(*
Nazwa:			FB_MoveRegister
Opis:			Blok przesuniecia rejestru formatek
Wersja:			v0.3 		
Data:			2018-11-16
Autor:			DP
Urzadzenia:		 
Konfiguracja:	
Info:
- Są dwa rejestry, wejściowy i wyjsciowy (struktury)
- Jezeli rejestr ma np. 6 elementów to za kazdym razem po wykryciu trigera program będzie
	1 wejściowy przesuwał na 1 wolny (nie ma formatki) wyjściowy
	kasował 1 rejestr wejściowy
	przesuwal rejetr wejsciowy 2 na 1(przeniesiony i skasowany), 3 na 2, 4 na 3, 5 na 4, 6 na 5 i kasowal 6wejsciowy
	tym sposobem po 6 trigerach caly rejestr wejsciowy powinien być na wyjsciowym
	np po 3 trigerach na wyjsciowym powinny byc zajete 1 do 3 i na wejsciowym 1 do 3
Błędy:
1 - nie wyszło z pętli for
2 - formatka już jest w rejestrze
Uwagi:
- 
Zmiany:
2018-09-18 Dodano sprawdzanie nasadek
2018-06-14 DP Pierwsza wersja
*)

FUNCTION_BLOCK FB_MoveRegisterCapControl
VAR_INPUT
	bFirstCycle:BOOL;					//Pierwszy cykl, zeby na początku nie wykrywało zbocza opadającego
	bTrigger :BOOL;						// Przesuniecie tablicy o jeden
	tTriggerFilterTimeOn:TIME:=T#0MS;	// Czas filtrowania wejścia Trigger na załączenie
	tTriggerFilterTimeOff:TIME:=T#0MS;	// Czas filtrowania wejścia Trigger na wyłączenie
	bTriggerBottle :BOOL;				// Zapisywanie czy jest butelka czy nie (jezeli kontrola wlączona)
	bWithBottleControl: BOOL;			// Włączona opcja kontroli butelek
	bWithCapControl:BOOL;				// Wlaczona kontrola nasadek
	bWithFormControlTrigerCounter:BOOL;	// Jezeku na trigercontrol nie ma formatki do przesunięcia to stwórz nową
	bNoKeepTryingMove:BOOL;				// Dalej przepisuj jezeli nie ma miejsca
	bTriggerCap: BOOL;					// Truger wykrycia nasadki
	bReset :BOOL;						// Czyszczenie tablic
	iEntranceArrayElements :UINT; 		// Wartość koncowa tablicy
	iExitArrayElements :UINT; 			// Wartość koncowa tablicy
	eClearPackageState :S_PackageState; // Czysty rejestr
END_VAR
VAR_IN_OUT
	eEntranceState :ARRAY [1..17] OF S_PackageState;	
	eExitState :ARRAY [1..17] OF S_PackageState;
	iBottleWithoutCap: INT;
	bKeepTryingMove :BOOL;		// Probuj dalej zapisać formatki aż się któraś zwolni
	bRFIDReaded :BOOL;
END_VAR

VAR_OUTPUT	
	bError :BOOL; 				// Błąd
	iError: UINT;				// Nr Błędu
	bTriggerDone :BOOL; 		// Wykonano przesunięcie

	bTriggerFilteredOUT:BOOL;	//Wyjscie przefiltrowanego sygnalu wejsciowego
END_VAR

VAR
	i:UINT;						// Zmienna w tablicy
	k:UINT;						// Pomocnicza zmienna do zapisywnia czy jest butelka
	rtbTrigger :R_TRIG;			// Reaguje na zbocze
	rtbTriggerBottle :R_TRIG;	// Reaguje na zbocze
	rtbReset :R_TRIG;			// Reaguje na zbocze
	TimerResetErrors :TON;		// Reset Błedu
	nFormCounter :UINT;					//Licznik formatek
	r1,r2:UINT;
	bBottlePresent: BOOL;				//Zmienna pomocnicza ze wykryto butelkę
	bCapPresent: BOOL;					//Zmienna pomocnicza ze wykryto butelkę
	j: UINT;
	tonTriggerFilterTimeOn: TON;
	bTriggerFiltered: BOOL;
	tofTriggerFilterTimeOff: TOF;
	fbTriggerFiltered: FB_InputFIlter;
	ftfbTriggerFiltered: F_TRIG;
	tpTrigger: TP;
END_VAR

//Filtrowanie sygnału wejściowego
fbTriggerFiltered		(bIN:= 	bTrigger AND bRFIDReaded,		tFilterTimeOn:=tTriggerFilterTimeOn,	tFilterTimeOff:=tTriggerFilterTimeOff);
tpTrigger				(IN:=bTrigger, 		PT:=T#10MS);
bTriggerFilteredOUT		:= fbTriggerFiltered.bOUT ;

//TRIGI I TIMERY
ftfbTriggerFiltered		(CLK:=	fbTriggerFiltered.bOUT, 	Q=>);

rtbReset 				(CLK := bReset, Q=>);
TimerResetErrors 		(IN:= bError, PT:=T#1000MS, Q=>);

//RESETOWANIE BLEDU
IF TimerResetErrors.Q THEN
	bError := FALSE;
END_IF

//KASOWANIE ZMIENNYCH
bTriggerDone := FALSE;

//JEZELI WLACZONO KONTROLE NASADEk TO NADPISUJ REJESTR CZY JEST BUTELKA 
IF bWithCapControl AND bTriggerCap AND NOT bKeepTryingMove THEN //Jezeli od wykrycia formatki liczy TIMER i wykryło butelke to wpisz do rejestru że jest butelka
	eEntranceState[1].bCapPutted := TRUE;
	eEntranceState[1].bCapOK := TRUE; eEntranceState[1].bBottlePresent:= TRUE;//Zmiana nowa
	bCapPresent := TRUE; // Wpisuje że jest butelka jezeli wystąpi sygnał podczas trwania czujnika formatki	
ELSIF bWithCapControl AND ftfbTriggerFiltered.Q AND NOT bCapPresent AND  NOT bKeepTryingMove AND bFirstCycle THEN
	eEntranceState[1].bCapPutted := TRUE;
	eEntranceState[1].bCapOK:= FALSE;
END_IF
//JEZELI WLACZONO SPRAWDZANIE FORMATEK Z TRIGERCOUNTER TO
IF  tpTrigger.Q AND NOT bKeepTryingMove AND bFirstCycle THEN //Zmiena UBL50, tworz tez nowa jak Trigger
	eEntranceState[1].bFormPresent := TRUE;
END_IF

//PRZESUNIECIE
IF iEntranceArrayElements < iExitArrayElements AND bFirstCycle THEN
	IF ftfbTriggerFiltered.Q OR bKeepTryingMove THEN
		bRFIDReaded		:= FALSE;
		bKeepTryingMove := FALSE;
		nFormCounter := 0;
		(*Do testów - jeszcze raz nadpisz jakby czujniki były przestawione LU205*)	
		IF bCapPresent THEN		
			eEntranceState[1].bCapPutted := TRUE;
			eEntranceState[1].bCapOK := TRUE; eEntranceState[1].bBottlePresent:= TRUE;//Zmiana nowa
			eEntranceState[1].bFormPresent := TRUE;
		END_IF
		(*Koniec Do testów - jeszcze raz nadpisz jakby czujniki były przestawione*)

		bBottlePresent := bCapPresent  := FALSE; 
		FOR i:= 1 TO iExitArrayElements-1 DO // SORTOWANIE
			IF NOT eExitState[i].bFormPresent THEN 
				eExitState[i] := eExitState[i+1];
				eExitState[i+1] := eClearPackageState;
			END_IF
		END_FOR
		FOR i := 1 TO iExitArrayElements DO
			IF  NOT eExitState[i].bFormPresent THEN  		// Jeżeli w rejestrze wyjściowym jest wolne miejsce to wpisz rejestr wejściowy
				eExitState[i] 		:= 	eEntranceState[1];			// Wpisz do rejestru dane np z [1] Buffor do [1,2,3,4,5,6] Package
				eEntranceState[1]	:=	eClearPackageState;		// Czyszczenie pierwszego rejestru wejściowego
				k:=i;										// Przepisywanie zmiennej pomocniczej
				bTriggerDone := TRUE;
				IF eExitState[i].bBottlePresent AND NOT eExitState[i].bCapOK THEN
					iBottleWithoutCap	:=	iBottleWithoutCap	+1;
				END_IF
				IF eExitState[i].bBottlePresent AND eExitState[i].bCapOK THEN
					iBottleWithoutCap	:=	0;	
				END_IF	
				IF NOT eExitState[i].bBottlePresent THEN
					iBottleWithoutCap	:=	0;	
				END_IF				
				EXIT;
				bError := TRUE;
				iError := 5;
			ELSE
				nFormCounter := nFormCounter + 1;
				bError := TRUE;
				iError := 6;
			END_IF
		END_FOR
		IF nFormCounter = iExitArrayElements THEN
			bKeepTryingMove:=NOT bNoKeepTryingMove;
		END_IF
	END_IF
END_IF

//CZYSZCZENIE REJESTRU WEJSCIOWEGO
IF rtbReset.Q THEN
	FOR r1 := 1 TO iEntranceArrayElements DO
		eEntranceState[r1] := eClearPackageState;
	END_FOR
	FOR r2 := 1 TO iExitArrayElements DO
		eExitState[r2] := eClearPackageState;
	END_FOR
	bKeepTryingMove :=FALSE;
	bTriggerDone := FALSE;
	nFormCounter := 0;
	bBottlePresent := bCapPresent := FALSE; 
	bError := FALSE;
	iError := 0;
END_IF

END_FUNCTION_BLOCK

(* stored: Version 1.1.0.1, ProductVersion 3.1.4026.13, FileIdentifier 02ff33d7c1e1b6a1c0f156e5d5aff0babdd9023b, FileSignature 647c9c777c942a8f77a578cf0d8726943087c07b7f24f5e4247d498e1210c067b9c241d41ac8fa590ea2b7de151d28e04e9adeefa224cf6dec89e85b8008fd50faa321ba86a8745d9d82c134ef2cdf35b79abd2ba8effa2dc56034c66afacb250629edf0a3ed9e2099ba08faa5d0849769744dd1e5de4d6183e5575aee4fccabc235ebcdc7820cb84d9e02597113051ba8c9ef0e8de1051bb65b881813fb7ad2ce70d804064aef501d8e2ce4adcf21b0b5646741ca13eb963cc1c89dd88611cbaa6f6d2f0aca5b2b8936afa683f8c890a102d51d77645c02642de67bbf64ea0cc00901b583cde48c740c3110b4792dfa4a4d168a7adcb3c5548cb1e94a869bc1
   POU FB_MoveRegisterCapControl: Id {816a9628-0bf9-42d6-90f2-05b524d2f084}, SpecialFunc None *)
